// TIA Portal project "babu_MicrowaveHMI" (V15)

(* hardware
DEVICE "S7-1200 station_1"  S7-1200 Station
   slot 0: "Rack_0"  S7-1200 Rack  Rack  V1.0
   slot 1: "PLC_1"  CPU 1214C DC/DC/DC  6ES7 214-1AG40-0XB0  V4.2
DEVICE "HMI_1"  KTP400 Basic PN
   slot 0: "HMI_1"  KTP400 Basic PN  6AV2 123-2DB03-0AX0  15.0.0.0
   slot 1: "HMI_RT_1"  KTP400 Basic PN  6AV2 123-2DB03-0AX0  15.0.0.0
   slot 5: "HMI_1.IE_CP_1"  PROFINET Interface  15.0.0.0
      slot 1: "PROFINET Interface_1"  PROFINET Interface
         slot 1: "Port_1"  Port
*)

// ===== PLC "PLC_1"  CPU 1214C DC/DC/DC =====

VAR_GLOBAL   // PLC tag table "Default tag table"
   "POWER ON PB" AT %M0.0 : Bool;
   "POWER ON PB MEM" AT %Q0.0 : Bool;
   "START PB" AT %M0.1 : Bool;
   "START PB MEM" AT %M0.2 : Bool;
   "COUNTS" AT %MW2 : Int;
   "COOK SECONDS" AT %MW4 : Int;
   "COOK SECS" AT %MD10 : DInt;
   "ROTATE COOKING MOTOR" AT %Q0.1 : Bool;
   "HEAT MICROWAVE" AT %Q0.2 : Bool;
   "COMPLETED ALARM" AT %Q0.3 : Bool;
   "COUNTER IP" AT %M0.3 : Bool;
   "COUNTER UP" AT %M0.4 : Bool;
   "COUNTER DOWN" AT %M0.5 : Bool;
END_VAR

// folder: System blocks/Program resources

DATA_BLOCK "IEC_Counter_0_DB"   // DB1
{ S7_Optimized_Access := 'TRUE' }
AUTHOR : Simatic
FAMILY : IEC
NAME : CNTR
VERSION : 1.0
// stored: InstanceOfName IEC_COUNTER
"IEC_COUNTER"
BEGIN
END_DATA_BLOCK

DATA_BLOCK "IEC_Timer_0_DB"   // DB2
{ S7_Optimized_Access := 'TRUE' }
AUTHOR : Simatic
FAMILY : IEC
NAME : IEC_TMR
VERSION : 1.0
// stored: InstanceOfName IEC_TIMER
"IEC_TIMER"
BEGIN
END_DATA_BLOCK

DATA_BLOCK "IEC_Timer_0_DB_1"   // DB3
{ S7_Optimized_Access := 'TRUE' }
AUTHOR : Simatic
FAMILY : IEC
NAME : IEC_TMR
VERSION : 1.0
// stored: InstanceOfName IEC_TIMER
"IEC_TIMER"
BEGIN
END_DATA_BLOCK

DATA_BLOCK "IEC_Timer_0_DB_2"   // DB4
{ S7_Optimized_Access := 'TRUE' }
AUTHOR : Simatic
FAMILY : IEC
NAME : IEC_TMR
VERSION : 1.0
// stored: InstanceOfName IEC_TIMER
"IEC_TIMER"
BEGIN
END_DATA_BLOCK

// folder: (top level)

ORGANIZATION_BLOCK "Main"   // OB1, LAD, ProgramCycle
TITLE = "Main Program Sweep (Cycle)"
{ S7_Optimized_Access := 'TRUE' }
VERSION : 0.1
   VAR_INPUT
      Initial_Call : Bool;   // Initial call of this OB
      Remanence : Bool;   // =True, if remanent data are available
   END_VAR
   VAR_TEMP   // added for the SCL form of the ladder/FBD networks
      _w1 : Bool;
   END_VAR
BEGIN

REGION Network 1
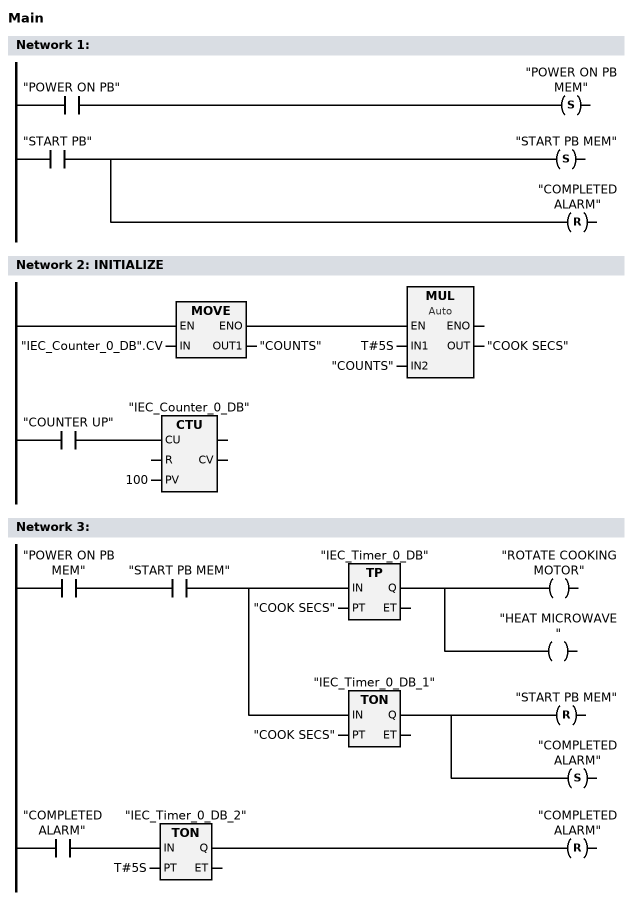
   RUNG wire#powerrail
      Contact( "POWER ON PB" )
      S_Coil( "POWER ON PB MEM" )
   END_RUNG
   RUNG wire#powerrail
      Contact( "START PB" )
      wire#w1
      S_Coil( "START PB MEM" )
   END_RUNG
   RUNG wire#w1
      R_Coil( "COMPLETED ALARM" )
   END_RUNG
   // the same network as SCL:
   IF "POWER ON PB" THEN "POWER ON PB MEM" := TRUE; END_IF;
   IF "START PB" THEN
       "START PB MEM" := TRUE;
       "COMPLETED ALARM" := FALSE;
   END_IF;
END_REGION

REGION Network 2: INITIALIZE
   "COUNTS" := "IEC_Counter_0_DB".CV;
   "COOK SECS" := T#5S * "COUNTS";
   "IEC_Counter_0_DB".CTU(CU := "COUNTER UP", PV := 100);
END_REGION

REGION Network 3
   #_w1 := "POWER ON PB MEM" AND "START PB MEM";
   "IEC_Timer_0_DB".TP(IN := #_w1, PT := "COOK SECS");
   "ROTATE COOKING MOTOR" := "IEC_Timer_0_DB".Q;
   "HEAT MICROWAVE" := "IEC_Timer_0_DB".Q;
   "IEC_Timer_0_DB_1".TON(IN := #_w1, PT := "COOK SECS");
   IF "IEC_Timer_0_DB_1".Q THEN
       "START PB MEM" := FALSE;
       "COMPLETED ALARM" := TRUE;
   END_IF;
   "IEC_Timer_0_DB_2".TON(IN := "COMPLETED ALARM", PT := T#5S);
   IF "IEC_Timer_0_DB_2".Q THEN "COMPLETED ALARM" := FALSE; END_IF;
END_REGION
END_ORGANIZATION_BLOCK